FUNCTION_BLOCK BfbSetterResetter
  (* Standard: 61499-2 *)
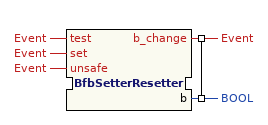
  EVENT_INPUT
    test;
    set;
    unsafe;
  END_EVENT
  EVENT_OUTPUT
    b_change WITH b;
  END_EVENT
  VAR_OUTPUT
    b : BOOL;
  END_VAR
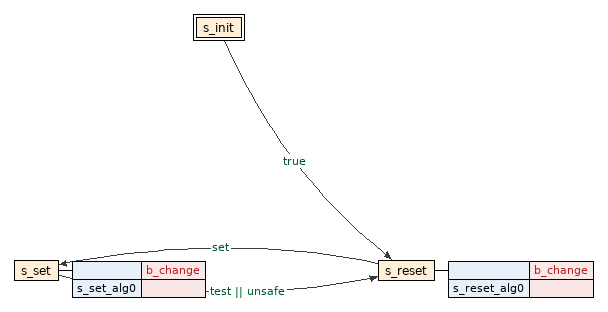
  EC_STATES
    s_init;
    s_reset : -> b_change, s_reset_alg0;
    s_set : -> b_change, s_set_alg0;
  END_STATES
  EC_TRANSITIONS
    s_init TO s_reset := true;
    s_reset TO s_set := set;
    s_set TO s_reset := test || unsafe;
  END_TRANSITIONS
  ALGORITHM s_reset_alg0 IN ST:
b := 0;
  END_ALGORITHM
  ALGORITHM s_set_alg0 IN ST:
b := 1;
  END_ALGORITHM
END_FUNCTION_BLOCK
